// TIA Portal V18 export
DATA_BLOCK "Function ConditionCheck without valve"   // DB135
{ S7_Optimized_Access := 'TRUE' }
VERSION : 0.1
// stored: AutoNumber true, DBAccessibleFromOPCUA true, IsOnlyStoredInLoadMemory false, IsRetainMemResEnabled false, IsWriteProtectedInAS false, MemoryReserve 100
   VAR
      "Control A" : Struct
         "start Condition Check" : Bool := FALSE;
         "Condition Check running" : Bool := FALSE;
         "stop Condition Check" : Bool := FALSE;
         "Condition Check Completed" : Bool := FALSE;
         "Pressure Setpoint" : Real := 0.0;
         Check_Time : DInt := 0;
         Pressure_tolerance : Real := 0.0;
         "Time tolerance" : Real := 0.0;
         "installtaion mode" : Bool := TRUE;
      END_STRUCT;
      "Control B" : Struct
         "start Condition Check" : Bool := FALSE;
         "Condition Check running" : Bool := FALSE;
         "stop Condition Check" : Bool := FALSE;
         "Condition Check Completed" : Bool := FALSE;
         "Pressure Setpoint" : Real := 0.0;
         Check_Time : DInt := 0;
         Pressure_tolerance : Real := 0.0;
         "Time tolerance" : Real := 0.0;
         "installation mode" : Bool := TRUE;
      END_STRUCT;
      "Output A" : Struct
         "ON pump" : Bool := FALSE;
         "running time" : Int := 0;
         "ON_inlet A" : Bool := FALSE;
         Pressure_OK : Bool := FALSE;
         Pressure_NOK : Bool := FALSE;
         Pressure_release_time : DInt := 0;
         Test_Fail : Bool := FALSE;
         "Test Pass" : Bool := FALSE;
      END_STRUCT;
      "Output B" : Struct
         "ON pump" : Bool := FALSE;
         "running time" : Int := 0;
         "ON_inlet B" : Bool := FALSE;
         Pressure_OK : Bool := FALSE;
         Pressure_NOK : Bool := FALSE;
         Pressure_release_time : DInt := 15;
         Test_Fail : Bool := FALSE;
         "Test Pass" : Bool := FALSE;
      END_STRUCT;
   END_VAR
   VAR RETAIN
      "Input A" : Struct
         "set time" : Int := 20;
         "set flowrate" : Real := 5.0;
         "Pressure Setpoint" : Real := 10.0;
         Check_Time : DInt := 15;
         Pressure_tolerance : Real := 3.0;
         PressurisingSP : Real := 5.0;
         Pressurisingtime : DInt := 45;
      END_STRUCT;
      "Input B" : Struct
         "set time" : Int := 20;
         "set flowrate" : Real := 5.0;
         "Pressure Setpoint" : Real := 10.0;
         Check_Time : DInt := 15;
         Pressure_tolerance : Real := 3.0;
         PressurisingSP : Real := 5.0;
         Pressurisingtime : DInt := 45;
      END_STRUCT;
   END_VAR
   VAR
      "start time" : DTL := DTL#1970-01-01-00:00:00;
      Stoptime : DTL := DTL#1970-01-01-00:00:00;
      "time in ms" : DInt := 0;
   END_VAR
   VAR RETAIN
      "Data A" : Struct
         "Pressure Achieved time @installation" : DInt := 92;
         "Pressure time @operation" : DInt := 0;
         "Pressure Achieved time @ operation" : Array[0..20] of DInt;
         "Leakage test pressure" : Real := 0.0;
         Test_Data : Array[1..20] of "Condition_Check";
         temp_Test_Data { S7_SetPoint := 'True'} : "Condition_Check";
      END_STRUCT;
      "Data B" : Struct
         "Pressure Achieved time @installation" : DInt := 71;
         "Pressure time @operation" : DInt := 0;
         "Pressure Achieved time @ operation" : Array[0..20] of DInt;
         "Leakage test pressure" : Real := 0.0;
         Test_Data : Array[1..20] of "Condition_Check";
         temp_Test_Data { S7_SetPoint := 'True'} : "Condition_Check";
      END_STRUCT;
   END_VAR
   VAR
      reset_FIFOA { S7_SetPoint := 'True'} : Bool := FALSE;
      reset_FIFOB : Bool := FALSE;
      Show_popupA : Bool := FALSE;
      Show_popupB : Bool := FALSE;
   END_VAR
   VAR RETAIN
      Condition_check_en : Bool := TRUE;
   END_VAR
   VAR
      start_revA_condcheck : Bool := FALSE;
      RevA_time : DInt := 3000;
   END_VAR
   VAR RETAIN
      RevA_flowrate : Real := 1.0;
   END_VAR
   VAR
      start_revB_condcheck : Bool := FALSE;
      RevB_time : DInt := 3000;
   END_VAR
   VAR RETAIN
      RevB_flowrate : Real := 1.0;
   END_VAR
BEGIN
   "Data A"."Pressure Achieved time @ operation"[0..20] := 0;
   "Data A".Test_Data[1].Date_time := DTL#2012-01-05-00:30:04.579546;
   "Data A".Test_Data[2].Date_time := DTL#2012-01-05-00:39:31.124577;
   "Data A".Test_Data[3..20].Date_time := DTL#1970-01-01-00:00:00;
   "Data A".Test_Data[1..2].Pressure_achieve_time := 92;
   "Data A".Test_Data[3..20].Pressure_achieve_time := 0;
   "Data A".Test_Data[1].Leakage_Pressure := 6.67;
   "Data A".Test_Data[2..20].Leakage_Pressure := 0.0;
   "Data A".Test_Data[1..2].Status := 2;
   "Data A".Test_Data[3..20].Status := 0;
   "Data A".temp_Test_Data.Date_time := DTL#1970-01-01-00:00:00;
   "Data A".temp_Test_Data.Pressure_achieve_time := 0;
   "Data A".temp_Test_Data.Leakage_Pressure := 0.0;
   "Data A".temp_Test_Data.Status := 0;
   "Data B"."Pressure Achieved time @ operation"[0..20] := 0;
   "Data B".Test_Data[1].Date_time := DTL#2012-01-05-00:42:23.319592;
   "Data B".Test_Data[2].Date_time := DTL#2012-01-05-00:50:51.810518;
   "Data B".Test_Data[3..20].Date_time := DTL#1970-01-01-00:00:00;
   "Data B".Test_Data[1].Pressure_achieve_time := 26;
   "Data B".Test_Data[2].Pressure_achieve_time := 71;
   "Data B".Test_Data[3..20].Pressure_achieve_time := 0;
   "Data B".Test_Data[1].Leakage_Pressure := 14.28;
   "Data B".Test_Data[2].Leakage_Pressure := 11.56;
   "Data B".Test_Data[3..20].Leakage_Pressure := 0.0;
   "Data B".Test_Data[1].Status := 2;
   "Data B".Test_Data[2].Status := 1;
   "Data B".Test_Data[3..20].Status := 0;
   "Data B".temp_Test_Data.Date_time := DTL#1970-01-01-00:00:00;
   "Data B".temp_Test_Data.Pressure_achieve_time := 0;
   "Data B".temp_Test_Data.Leakage_Pressure := 0.0;
   "Data B".temp_Test_Data.Status := 0;
END_DATA_BLOCK
